{attribute 'qualified_only'}
{attribute 'strict'}
TYPE LightCurtainStatus :
(
	UNKNOWN := 0, UNBLOCKED := 1, BLOCKED := 2
);
END_TYPE

(* stored: Version 1.1.0.1, ProductVersion 3.1.4024.12
   DUT LightCurtainStatus: Id {d1037462-91c9-448d-9a1b-5410d942a307} *)
